TYPE ST_Logging :
STRUCT
     bError		: BOOL;
     nErrorId  	: UDINT;
END_STRUCT
END_TYPE

(* stored: Version 1.1.0.1
   DUT ST_Logging: Id {47a76e17-b64e-4575-a0bd-28a48da1e4a5} *)
